FUNCTION_BLOCK FB_MessageDynamique
// Allows to create dynamic messages in order to add variable to a string
VAR_INPUT
	
	InMessage	: ST_ValuesAlarms;
	InNbparam	: SINT;
END_VAR
VAR_OUTPUT
	OutMessage	: STRING(150);
END_VAR
VAR
	Valeur  	: STRING(10); // Nom de la balise a tester
	P	    	: INT;		 // Pos de la balise dans une chaine de caractere 
	i,j			: SINT;		// Compteur incrémental
	Temp		: String(150);
END_VAR

Temp:=InMessage.Message;
FOR i:=1 TO InNbparam DO
	IF InMessage.Ax_ParamB[i]<>0 THEN
		Valeur := BOOL_TO_STRING(InMessage.Ax_ParamB[i]^);
		P      := FIND(Temp,concat('<Balise_B',INT_TO_STRING(i)));
		IF P >0 THEN
			Temp:=Replace(Temp,Valeur,10,P);
		ELSE
			EXIT;
		END_IF
	END_IF
END_FOR

FOR j:=1 TO InNbparam DO
	IF InMessage.Ax_ParamI[j]<>0 THEN
		Valeur := SINT_TO_STRING(InMessage.Ax_ParamI[j]^);
		P      := FIND(temp,concat('<Balise_I',INT_TO_STRING(j)));
		IF P >0 THEN
			Temp:=Replace(temp,Valeur,10,P);
		ELSE
			EXIT;
		END_IF
	END_IF
END_FOR
OutMessage:=Temp;

END_FUNCTION_BLOCK

(* stored: Version 1.1.0.1, ProductVersion 3.1.4024.6
   POU FB_MessageDynamique: Id {51920e01-377f-461f-a1d1-fce62e2529a9}, SpecialFunc None *)
